SYSTEM PNP_MVCLF (* Pick & Place Model/View with FBD Controller *)
  (* Standard: IEC 61499; Classification: Simulation; ApplicationDomain: Assembly; Function: Control; Type: Pick & Place *)
  (* Version 1.1, 2007-09-24, JHC, Holobloc Inc, Simplified PNP.CLOCK. *)
  (* Version 1.0, 2006-09-18, JHC, Holobloc Inc, Moved CNV_CTL to PNP device. *)
  (* Version 0.9, 2006-09-16, JHC, Holobloc Inc, Cleaned up CONTROL.CONVEYOR; moved CNV_LOAD to PNP.CONVEYOR. *)
  (* Version 0.8, 2006-09-16, JHC, Holobloc Inc, Updated for PNP_CTL_LD as SimpleFB. *)
  (* Version 0.7, 2006-07-07, JHC, Holobloc Inc, Separated PRESENT/LOADED sensors; revised controller; changed HMI layout. *)
  (* Version 0.6, 2006-07-04, JHC, Holobloc Inc, Added S0 activation delay in PNP.XY. *)
  (* Version 0.5, 2006-07-03, JHC, Holobloc Inc, Added simulation logic to LOAD only when PNP is already unloaded. *)
  (* Version 0.4, 2006-07-03, JHC, Holobloc Inc, Added STOP button and logic in MODE_CTL. *)
  (* Version 0.3, 2006-07-03, JHC, Holobloc Inc, Added MAGNET ON/OFF cycle to PNP.CLOCK to init simulation correctly. *)
  (* Version 0.2, 2006-06-29, JHC, Holobloc Inc, Added simulation logic to LOAD only in HOME position. *)
  (* Version 0.1, 2006-06-27, JHC, Holobloc Inc, Added S0 simulation logic. *)
  (* Version 0.0, 2006-06-25, JHC, Holobloc Inc *)
  DEVICE PNP : FRAME_DEVICE(BOUNDS := [475,100,160,230])
    RESOURCE CLOCK : EMB_RES
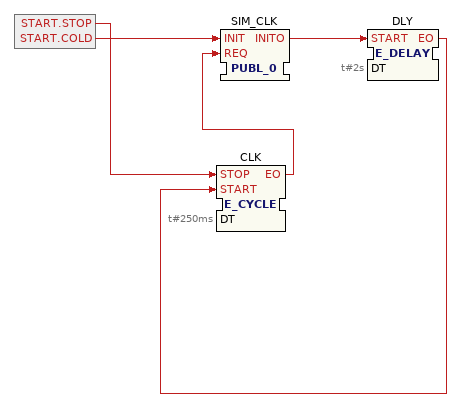
      FBS
        CLK : E_CYCLE(DT := t#250ms);
        SIM_CLK : PUBL_0;
        DLY : E_DELAY(DT := t#2s); (* Wait for View startup *)
      END_FBS
      EVENT_CONNECTIONS
        START.STOP TO CLK.STOP;
        START.COLD TO SIM_CLK.INIT;
        SIM_CLK.INITO TO DLY.START;
        DLY.EO TO CLK.START;
        CLK.EO TO SIM_CLK.REQ;
      END_CONNECTIONS
    END_RESOURCE
    RESOURCE CONVEYOR : EMB_RES
      FBS
        CNV : CNV_MDLL(VF := 10);
        PRESENT : PUBL_1; (* Workpiece present at end of conveyor *)
        S0_SENSE : V_SENSE(REFSTYLE := VSTYLE#BALL);
        CNV_UNLD : SUBL_0;
        CNV_LD : SUBL_0;
        CNV_LOAD : LOADL(STYLE := VSTYLE#BALL, WKPC := [255,255,0], ID := "CNV_LOAD");
      END_FBS
      EVENT_CONNECTIONS
        CNV.INDS TO S0_SENSE.SENSE;
        S0_SENSE.IND TO PRESENT.REQ;
        CNV.INITO TO PRESENT.INIT;
        START.COLD TO CNV_UNLD.INIT;
        CNV_UNLD.INITO TO CNV.INIT;
        CNV_UNLD.IND TO CNV.UNLD;
        PRESENT.INITO TO CNV_LD.INIT;
        CNV_LD.INITO TO CNV_LOAD.INIT;
        CNV_LD.IND TO CNV_LOAD.REQ;
      END_CONNECTIONS
      DATA_CONNECTIONS
        CNV.END TO S0_SENSE.PRESENT;
        CNV.STYLO TO S0_SENSE.STYLE;
        S0_SENSE.Q TO PRESENT.SD_1;
      END_CONNECTIONS
    END_RESOURCE
    RESOURCE CNV_CTL : PANEL_RESOURCE(ROWS := 2, COLS := 2)
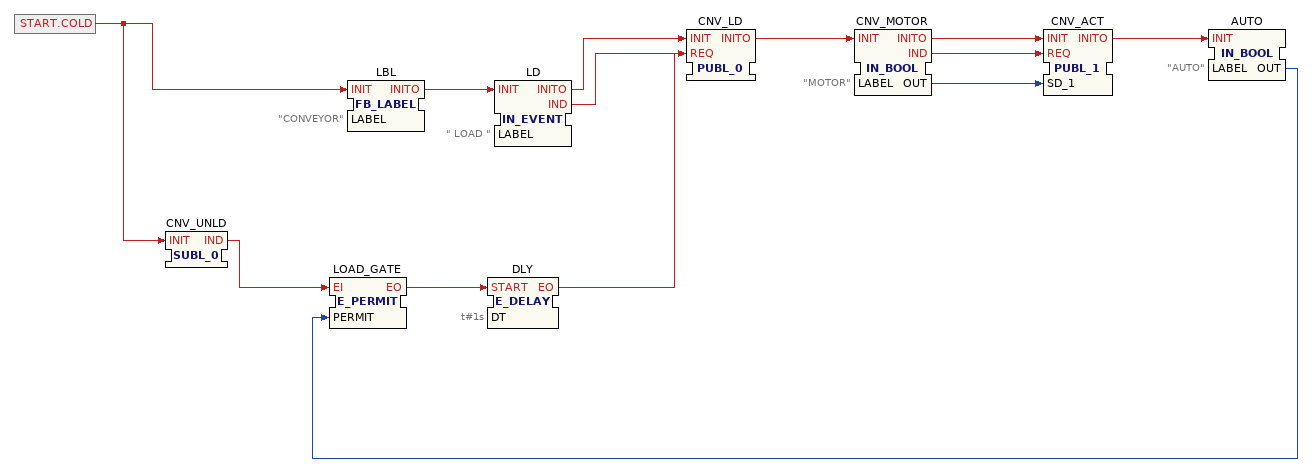
      FBS
        LD : IN_EVENT(LABEL := "    LOAD    ");
        CNV_LD : PUBL_0;
        CNV_MOTOR : IN_BOOL(LABEL := "MOTOR");
        CNV_ACT : PUBL_1;
        CNV_UNLD : SUBL_0; (* Conveyor unloaded by Magnet *)
        AUTO : IN_BOOL(LABEL := "AUTO"); (* Conveyor auto-reload *)
        LBL : FB_LABEL(LABEL := "CONVEYOR");
        DLY : E_DELAY(DT := t#1s); (* Breaks unload/reload loop *)
        LOAD_GATE : E_PERMIT;
      END_FBS
      EVENT_CONNECTIONS
        LD.INITO TO CNV_LD.INIT;
        LD.IND TO CNV_LD.REQ;
        CNV_LD.INITO TO CNV_MOTOR.INIT;
        CNV_MOTOR.INITO TO CNV_ACT.INIT;
        CNV_MOTOR.IND TO CNV_ACT.REQ;
        CNV_ACT.INITO TO AUTO.INIT;
        START.COLD TO LBL.INIT;
        LBL.INITO TO LD.INIT;
        DLY.EO TO CNV_LD.REQ;
        START.COLD TO CNV_UNLD.INIT;
        CNV_UNLD.IND TO LOAD_GATE.EI;
        LOAD_GATE.EO TO DLY.START;
      END_CONNECTIONS
      DATA_CONNECTIONS
        CNV_MOTOR.OUT TO CNV_ACT.SD_1;
        AUTO.OUT TO LOAD_GATE.PERMIT;
      END_CONNECTIONS
    END_RESOURCE
    RESOURCE XY : EMB_RES
      FBS
        PNP : XY_MDLL(UI_ID := "FAULT");
        MAGNET : SUBL_1;
        LD_GATE1 : FB_AND;
        CNV_UNLD : PUBL_0;
        PNP_MT : FB_NOT; (* No workpiece loaded to PNP unit *)
        LD_GATE2 : FB_AND;
        UNLD : E_F_TRIG;
        PRESENT : SUBL_1;
        LD_GATE3 : FB_AND;
        LD_GATE4 : FB_AND;
        LD_TRIG : E_R_TRIG;
        PNP_LOAD : LOADL(STYLE := VSTYLE#BALL, WKPC := [255,255,0], ID := "PNP_LOAD");
      END_FBS
      EVENT_CONNECTIONS
        MAGNET.IND TO UNLD.EI;
        UNLD.EO TO PNP.UNLD;
        PNP.IND TO PNP_MT.REQ;
        PNP_MT.CNF TO LD_GATE1.REQ;
        LD_GATE1.CNF TO LD_GATE2.REQ;
        PRESENT.IND TO LD_GATE3.REQ;
        MAGNET.IND TO LD_GATE4.REQ;
        LD_GATE3.CNF TO LD_GATE4.REQ;
        LD_GATE4.CNF TO LD_TRIG.EI;
        START.COLD TO PNP.INIT;
        MAGNET.INITO TO PNP_LOAD.INIT;
        LD_TRIG.EO TO PNP_LOAD.REQ;
        PNP_LOAD.INITO TO CNV_UNLD.INIT;
        PNP_LOAD.CNF TO CNV_UNLD.REQ;
        LD_GATE2.CNF TO LD_GATE3.REQ;
        PNP.INITO TO MAGNET.INIT;
        PNP.INITO TO PRESENT.INIT;
      END_CONNECTIONS
      DATA_CONNECTIONS
        MAGNET.RD_1 TO UNLD.QI;
        PNP.HOMEX TO LD_GATE1.IN2;
        PNP.HOMEY TO LD_GATE2.IN2;
        LD_GATE1.OUT TO LD_GATE2.IN1;
        PRESENT.RD_1 TO LD_GATE3.IN1;
        LD_GATE2.OUT TO LD_GATE3.IN2;
        LD_GATE4.OUT TO LD_TRIG.QI;
        PNP.LOADED TO PNP_MT.IN;
        PNP_MT.OUT TO LD_GATE1.IN1;
        LD_GATE3.OUT TO LD_GATE4.IN1;
        MAGNET.RD_1 TO LD_GATE4.IN2;
      END_CONNECTIONS
    END_RESOURCE
    RESOURCE VIEW : VIEW_PANEL(DIA := 25, SIZE := [6,5], VERTICAL := 0)
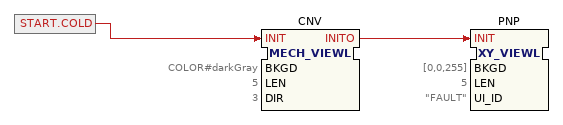
      FBS
        PNP : XY_VIEWL(BKGD := [0,0,255], LEN := 5, UI_ID := "FAULT");
        CNV : MECH_VIEWL(BKGD := COLOR#darkGray, LEN := 5, DIR := 3); (* Conveyor *)
      END_FBS
      EVENT_CONNECTIONS
        START.COLD TO CNV.INIT;
        CNV.INITO TO PNP.INIT;
      END_CONNECTIONS
    END_RESOURCE
  END_DEVICE
  DEVICE CONTROL : FRAME_DEVICE(BOUNDS := [100,100,375,180], GRID := [1,4]) (* Control + HMI *)
    RESOURCE MODE_CTL : PANEL_RESOURCE
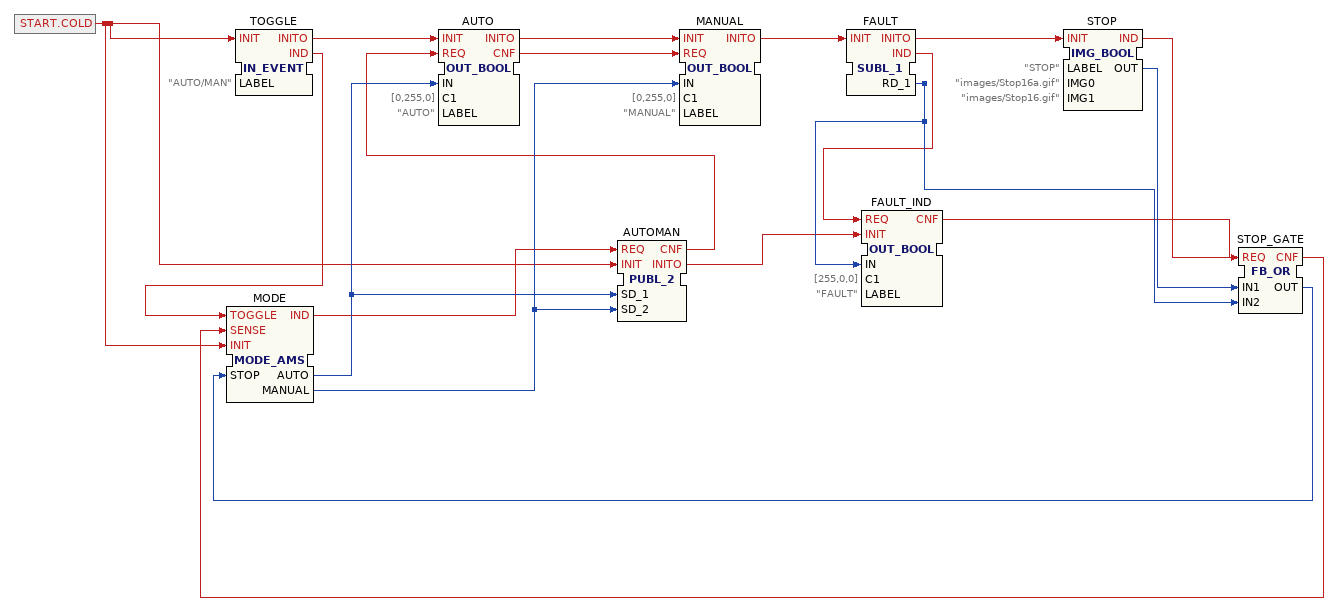
      FBS
        FAULT_IND : OUT_BOOL(C1 := [255,0,0], LABEL := "FAULT");
        FAULT : SUBL_1;
        AUTOMAN : PUBL_2;
        MODE : MODE_AMS;
        TOGGLE : IN_EVENT(LABEL := "AUTO/MAN");
        AUTO : OUT_BOOL(C1 := [0,255,0], LABEL := "AUTO");
        MANUAL : OUT_BOOL(C1 := [0,255,0], LABEL := "MANUAL");
        STOP : IMG_BOOL(LABEL := "STOP", IMG0 := "images/Stop16a.gif", IMG1 := "images/Stop16.gif");
        STOP_GATE : FB_OR;
      END_FBS
      EVENT_CONNECTIONS
        START.COLD TO TOGGLE.INIT;
        TOGGLE.INITO TO AUTO.INIT;
        AUTO.INITO TO MANUAL.INIT;
        AUTO.CNF TO MANUAL.REQ;
        MODE.IND TO AUTOMAN.REQ;
        TOGGLE.IND TO MODE.TOGGLE;
        AUTOMAN.CNF TO AUTO.REQ;
        STOP.IND TO STOP_GATE.REQ;
        MANUAL.INITO TO FAULT.INIT;
        FAULT.INITO TO STOP.INIT;
        FAULT.IND TO FAULT_IND.REQ;
        FAULT_IND.CNF TO STOP_GATE.REQ;
        STOP_GATE.CNF TO MODE.SENSE;
        START.COLD TO AUTOMAN.INIT;
        AUTOMAN.INITO TO FAULT_IND.INIT;
        START.COLD TO MODE.INIT;
      END_CONNECTIONS
      DATA_CONNECTIONS
        FAULT.RD_1 TO FAULT_IND.IN;
        MODE.AUTO TO AUTOMAN.SD_1;
        MODE.MANUAL TO AUTOMAN.SD_2;
        MODE.AUTO TO AUTO.IN;
        MODE.MANUAL TO MANUAL.IN;
        STOP.OUT TO STOP_GATE.IN1;
        FAULT.RD_1 TO STOP_GATE.IN2;
        STOP_GATE.OUT TO MODE.STOP;
      END_CONNECTIONS
    END_RESOURCE
    RESOURCE AUTO_CTL : EMB_RES
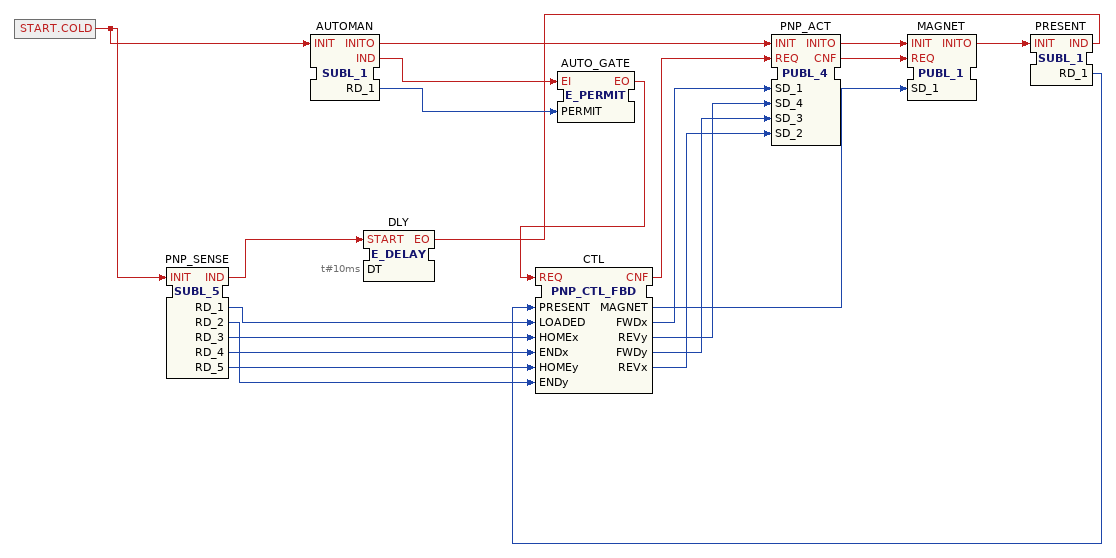
      FBS
        CTL : PNP_CTL_FBD;
        AUTOMAN : SUBL_1;
        MAGNET : PUBL_1;
        PNP_ACT : PUBL_4;
        PNP_SENSE : SUBL_5;
        PRESENT : SUBL_1;
        DLY : E_DELAY(DT := t#10ms); (* Breaks magnet/loader loop *)
        AUTO_GATE : E_PERMIT;
      END_FBS
      EVENT_CONNECTIONS
        START.COLD TO AUTOMAN.INIT;
        START.COLD TO PNP_SENSE.INIT;
        AUTOMAN.INITO TO PNP_ACT.INIT;
        CTL.CNF TO PNP_ACT.REQ;
        PNP_ACT.INITO TO MAGNET.INIT;
        PNP_ACT.CNF TO MAGNET.REQ;
        MAGNET.INITO TO PRESENT.INIT;
        PNP_SENSE.IND TO DLY.START;
        AUTOMAN.IND TO AUTO_GATE.EI;
        PRESENT.IND TO AUTO_GATE.EI;
        DLY.EO TO AUTO_GATE.EI;
        AUTO_GATE.EO TO CTL.REQ;
      END_CONNECTIONS
      DATA_CONNECTIONS
        CTL.MAGNET TO MAGNET.SD_1;
        CTL.FWDx TO PNP_ACT.SD_1;
        CTL.REVy TO PNP_ACT.SD_4;
        CTL.FWDy TO PNP_ACT.SD_3;
        CTL.REVx TO PNP_ACT.SD_2;
        PRESENT.RD_1 TO CTL.PRESENT;
        PNP_SENSE.RD_1 TO CTL.LOADED;
        PNP_SENSE.RD_2 TO CTL.HOMEx;
        PNP_SENSE.RD_3 TO CTL.ENDx;
        PNP_SENSE.RD_4 TO CTL.HOMEy;
        PNP_SENSE.RD_5 TO CTL.ENDy;
        AUTOMAN.RD_1 TO AUTO_GATE.PERMIT;
      END_CONNECTIONS
    END_RESOURCE
    RESOURCE ACTUATORS : PANEL_RESOURCE
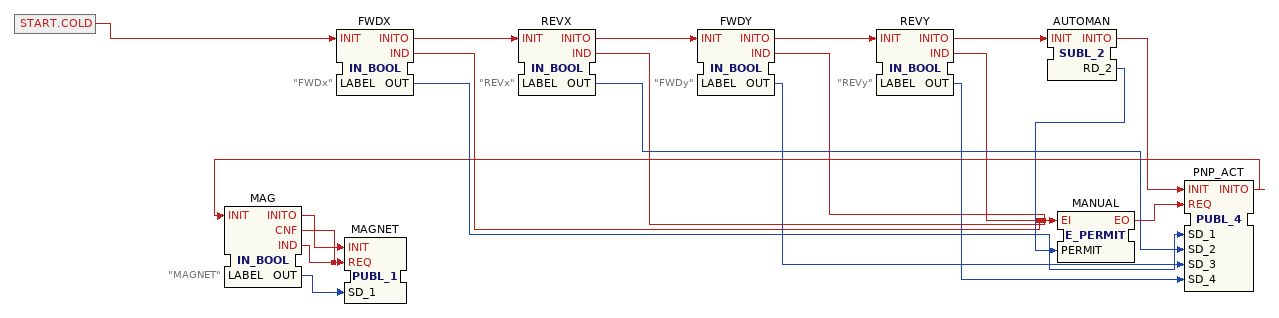
      FBS
        PNP_ACT : PUBL_4;
        FWDX : IN_BOOL(LABEL := "FWDx");
        REVX : IN_BOOL(LABEL := "REVx");
        FWDY : IN_BOOL(LABEL := "FWDy");
        REVY : IN_BOOL(LABEL := "REVy");
        MAG : IN_BOOL(LABEL := "MAGNET");
        MAGNET : PUBL_1;
        AUTOMAN : SUBL_2;
        MANUAL : E_PERMIT;
      END_FBS
      EVENT_CONNECTIONS
        START.COLD TO FWDX.INIT;
        FWDX.INITO TO REVX.INIT;
        REVX.INITO TO FWDY.INIT;
        FWDY.INITO TO REVY.INIT;
        MAG.INITO TO MAGNET.INIT;
        MAG.CNF TO MAGNET.REQ;
        MAG.IND TO MAGNET.REQ;
        PNP_ACT.INITO TO MAG.INIT;
        REVY.INITO TO AUTOMAN.INIT;
        AUTOMAN.INITO TO PNP_ACT.INIT;
        MANUAL.EO TO PNP_ACT.REQ;
        REVY.IND TO MANUAL.EI;
        FWDY.IND TO MANUAL.EI;
        REVX.IND TO MANUAL.EI;
        FWDX.IND TO MANUAL.EI;
      END_CONNECTIONS
      DATA_CONNECTIONS
        FWDX.OUT TO PNP_ACT.SD_1;
        REVX.OUT TO PNP_ACT.SD_2;
        FWDY.OUT TO PNP_ACT.SD_3;
        REVY.OUT TO PNP_ACT.SD_4;
        MAG.OUT TO MAGNET.SD_1;
        AUTOMAN.RD_2 TO MANUAL.PERMIT;
      END_CONNECTIONS
    END_RESOURCE
    RESOURCE ACT_STATE : PANEL_RESOURCE
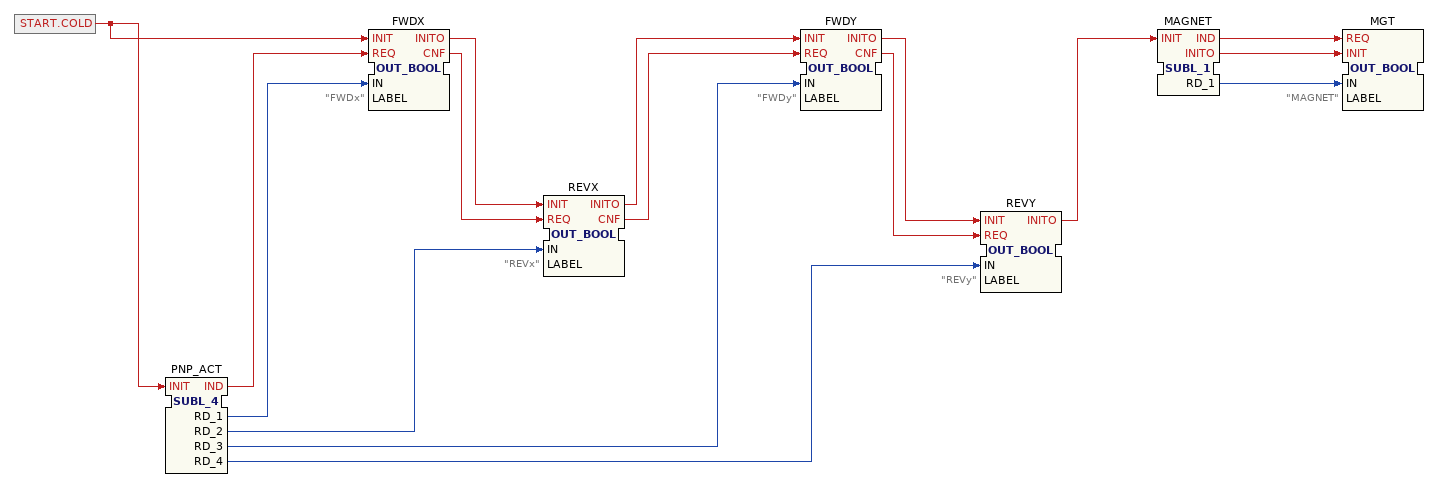
      FBS
        FWDX : OUT_BOOL(LABEL := "FWDx");
        REVX : OUT_BOOL(LABEL := "REVx");
        FWDY : OUT_BOOL(LABEL := "FWDy");
        REVY : OUT_BOOL(LABEL := "REVy");
        MGT : OUT_BOOL(LABEL := "MAGNET");
        PNP_ACT : SUBL_4;
        MAGNET : SUBL_1;
      END_FBS
      EVENT_CONNECTIONS
        START.COLD TO FWDX.INIT;
        FWDX.INITO TO REVX.INIT;
        REVX.INITO TO FWDY.INIT;
        FWDY.INITO TO REVY.INIT;
        START.COLD TO PNP_ACT.INIT;
        PNP_ACT.IND TO FWDX.REQ;
        FWDX.CNF TO REVX.REQ;
        REVX.CNF TO FWDY.REQ;
        FWDY.CNF TO REVY.REQ;
        MAGNET.IND TO MGT.REQ;
        REVY.INITO TO MAGNET.INIT;
        MAGNET.INITO TO MGT.INIT;
      END_CONNECTIONS
      DATA_CONNECTIONS
        PNP_ACT.RD_1 TO FWDX.IN;
        PNP_ACT.RD_2 TO REVX.IN;
        PNP_ACT.RD_3 TO FWDY.IN;
        PNP_ACT.RD_4 TO REVY.IN;
        MAGNET.RD_1 TO MGT.IN;
      END_CONNECTIONS
    END_RESOURCE
    RESOURCE SENSORS : PANEL_RESOURCE
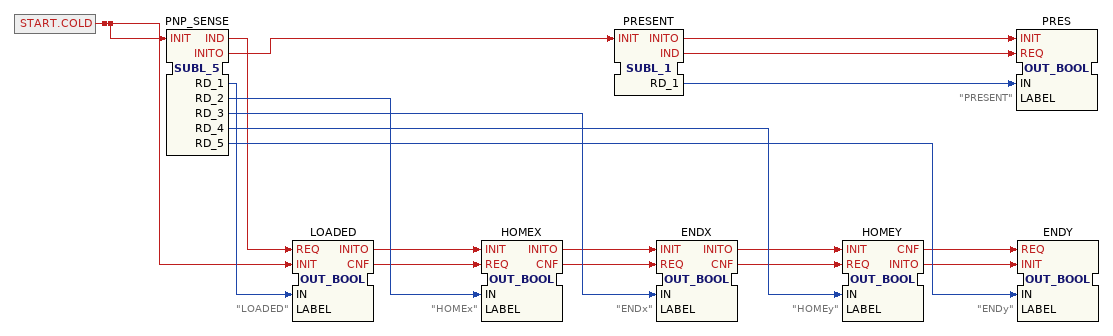
      FBS
        PNP_SENSE : SUBL_5;
        HOMEX : OUT_BOOL(LABEL := "HOMEx");
        ENDX : OUT_BOOL(LABEL := "ENDx");
        HOMEY : OUT_BOOL(LABEL := "HOMEy");
        ENDY : OUT_BOOL(LABEL := "ENDy");
        LOADED : OUT_BOOL(LABEL := "LOADED");
        PRESENT : SUBL_1;
        PRES : OUT_BOOL(LABEL := "PRESENT");
      END_FBS
      EVENT_CONNECTIONS
        START.COLD TO PNP_SENSE.INIT;
        HOMEX.INITO TO ENDX.INIT;
        HOMEX.CNF TO ENDX.REQ;
        ENDX.INITO TO HOMEY.INIT;
        HOMEY.CNF TO ENDY.REQ;
        HOMEY.INITO TO ENDY.INIT;
        ENDX.CNF TO HOMEY.REQ;
        LOADED.INITO TO HOMEX.INIT;
        PNP_SENSE.IND TO LOADED.REQ;
        LOADED.CNF TO HOMEX.REQ;
        PNP_SENSE.INITO TO PRESENT.INIT;
        PRESENT.INITO TO PRES.INIT;
        PRESENT.IND TO PRES.REQ;
        START.COLD TO LOADED.INIT;
      END_CONNECTIONS
      DATA_CONNECTIONS
        PNP_SENSE.RD_1 TO LOADED.IN;
        PNP_SENSE.RD_2 TO HOMEX.IN;
        PNP_SENSE.RD_3 TO ENDX.IN;
        PNP_SENSE.RD_4 TO HOMEY.IN;
        PNP_SENSE.RD_5 TO ENDY.IN;
        PRESENT.RD_1 TO PRES.IN;
      END_CONNECTIONS
    END_RESOURCE
  END_DEVICE
END_SYSTEM
